FUNCTION_BLOCK PressureGradient
VAR_INPUT
	TotalVolume: LREAL;
	BulkModulus: LREAL;
	FlowrateIn: LREAL;
	FlowrateOut: LREAL;
END_VAR
VAR_OUTPUT
	PressureGradientBar : LREAL;
	PressureGradientPascal : LREAL;
	PressureBar : LREAL;
	PressurePascal : LREAL;
END_VAR
VAR
	ssMethodType : SINT := 1; 
	fbPressureBar : DiscreteIntegrator;
END_VAR


(* Outputs for Atomic SubSystem: '<Root>/PressureGradient' *)
(* Outport: '<Root>/PressureGradientb' incorporates:
 *  Gain: '<S1>/Conv.2'
 *  Product: '<S1>/Product'
 *  Product: '<S1>/Product1'
 *  Sum: '<S1>/Sum' *)
 
//PressureGradient in [Bar/s]
PressureGradientBar := ((FlowrateIn - FlowrateOut) * 1.6666666666666667E-5) * (Param.BulkModulus / TotalVolume);
(* End of Outputs for SubSystem: '<Root>/PressureGradient' *)

//Multiplies to get [Pascal/s]
PressureGradientPascal := PressureGradientBar*1E5; 

//Pressure in [Pascal]
fbPressureBar(
	ssMethodType := ssMethodType,
	In1 := PressureGradientBar,
	Out1 => PressureBar
	);

//Pressure in [Bar]
PressurePascal := PressureBar*1E5;

END_FUNCTION_BLOCK

(* stored: Version 1.1.0.1, ProductVersion 3.1.4024.9
   POU PressureGradient: Id {0ae25e94-6017-429e-9462-38875999b492}, SpecialFunc None *)
